(* PLC project mode, Dassault Systèmes ControlBuild 2024x Refresh1 *)
(* stored: creationDateTime 2024-04-12T14:05:56-01:00 *)

FUNCTION_BLOCK copie_batch.mode
  VAR_INPUT
    powerUp : BOOL := false;
    emergencyStop : BOOL := false;
    manualSwitch : BOOL := false;
    autoSwitch : BOOL := false;
    startCyclePB : BOOL := false;
    endCyclePB : BOOL := false;
  END_VAR
  VAR_INPUT
    acknowledgePB : BOOL := false;
    cycleEnd : BOOL := false;
    generalFault : BOOL := false;
  END_VAR
  VAR_OUTPUT
    live : BOOL := false;
  END_VAR
  VAR_OUTPUT
    autoMode : BOOL := false;
    manualMode : BOOL := false;
  END_VAR
  VAR_OUTPUT
    cycleInProgress : BOOL := false;
    endCycleRequest : BOOL := false;
  END_VAR
  VAR
    emergencyStopState : BOOL := false;
  END_VAR
  VAR  (* added by the conversion: wires and edge detectors of the diagram *)
    R_TRIG1 : R_TRIG;
    F_TRIG2 : F_TRIG;
  END_VAR

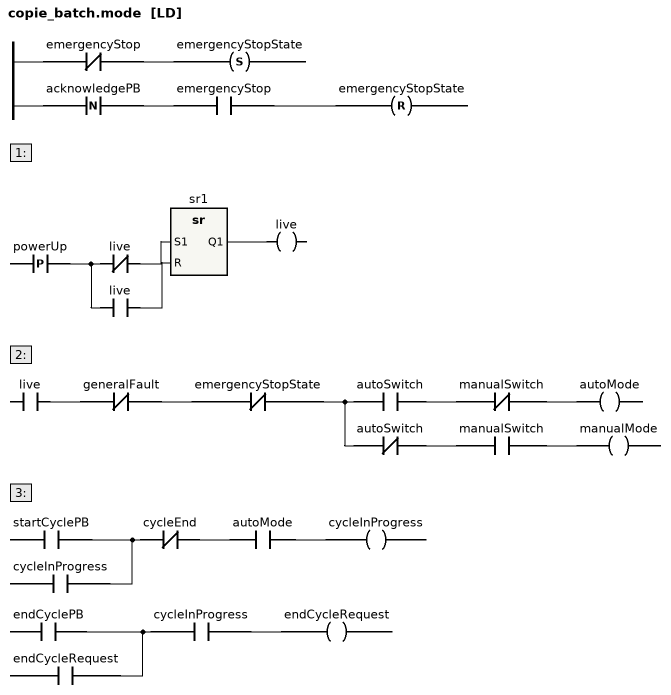
(* LD diagram, written out as Structured Text *)
1:
R_TRIG1(CLK := powerUp);
sr1(S1 := R_TRIG1.Q AND NOT live, R := R_TRIG1.Q AND live);
live := sr1.Q1;
2:
IF NOT emergencyStop THEN emergencyStopState := TRUE; END_IF;
F_TRIG2(CLK := acknowledgePB);
IF F_TRIG2.Q AND emergencyStop THEN emergencyStopState := FALSE; END_IF;
autoMode := live AND NOT generalFault AND NOT emergencyStopState AND autoSwitch AND NOT manualSwitch;
manualMode := live AND NOT generalFault AND NOT emergencyStopState AND NOT autoSwitch AND manualSwitch;
3:
cycleInProgress := (cycleInProgress OR startCyclePB) AND NOT cycleEnd AND autoMode;
endCycleRequest := (endCyclePB OR endCycleRequest) AND cycleInProgress;
END_FUNCTION_BLOCK
